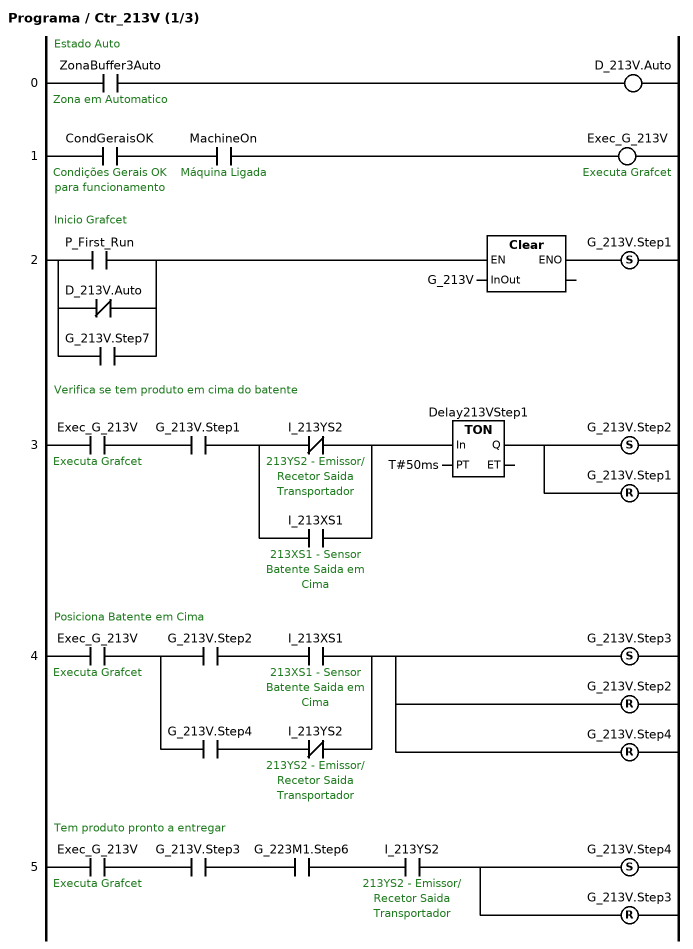
(* [picture p48: Programa / Ctr_213V, rungs 0-5] *)
(* Rung 0: Estado Auto *)
D_213V.Auto := ZonaBuffer3Auto;
(* Rung 1 *)
Exec_G_213V := CondGeraisOK AND MachineOn;
(* Rung 2: Inicio Grafcet *)
_p80 := P_First_Run OR NOT D_213V.Auto OR G_213V.Step7;
IF _p80 THEN
    Clear(InOut := G_213V);
    G_213V.Step1 := TRUE;
END_IF;
(* Rung 3: Verifica se tem produto em cima do batente *)
Delay213VStep1(In := Exec_G_213V AND G_213V.Step1 AND (NOT I_213YS2 OR I_213XS1), PT := T#50ms);
IF Delay213VStep1.Q THEN
    G_213V.Step2 := TRUE;
    G_213V.Step1 := FALSE;
END_IF;
(* Rung 4: Posiciona Batente em Cima *)
_p81 := Exec_G_213V AND ((G_213V.Step2 AND I_213XS1) OR (G_213V.Step4 AND NOT I_213YS2));
IF _p81 THEN
    G_213V.Step3 := TRUE;
    G_213V.Step2 := FALSE;
    G_213V.Step4 := FALSE;
END_IF;
(* Rung 5: Tem produto pronto a entregar *)
_p82 := Exec_G_213V AND G_213V.Step3 AND G_223M1.Step6 AND I_213YS2;
IF _p82 THEN
    G_213V.Step4 := TRUE;
    G_213V.Step3 := FALSE;
END_IF;

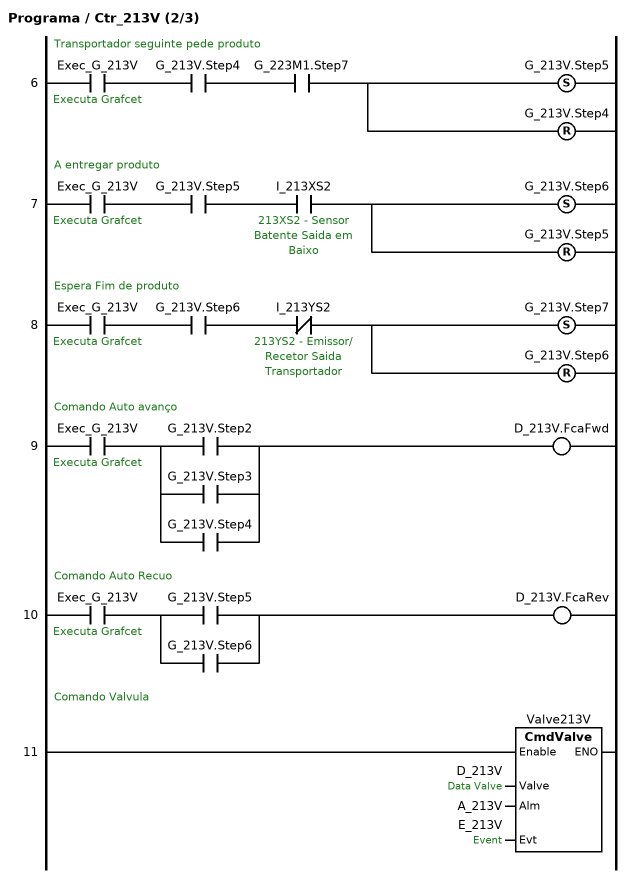
(* Rung 6: Transportador seguinte pede produto *)
_p83 := Exec_G_213V AND G_213V.Step4 AND G_223M1.Step7;
IF _p83 THEN
    G_213V.Step5 := TRUE;
    G_213V.Step4 := FALSE;
END_IF;
(* Rung 7: A entregar produto *)
_p84 := Exec_G_213V AND G_213V.Step5 AND I_213XS2;
IF _p84 THEN
    G_213V.Step6 := TRUE;
    G_213V.Step5 := FALSE;
END_IF;
(* Rung 8: Espera Fim de produto *)
_p85 := Exec_G_213V AND G_213V.Step6 AND NOT I_213YS2;
IF _p85 THEN
    G_213V.Step7 := TRUE;
    G_213V.Step6 := FALSE;
END_IF;
(* Rung 9: Comando Auto avanço *)
D_213V.FcaFwd := Exec_G_213V AND (G_213V.Step2 OR G_213V.Step3 OR G_213V.Step4);
(* Rung 10: Comando Auto Recuo *)
D_213V.FcaRev := Exec_G_213V AND (G_213V.Step5 OR G_213V.Step6);
(* Rung 11: Comando Valvula *)
Valve213V(Enable := TRUE, Valve := D_213V, Alm := A_213V, Evt := E_213V);

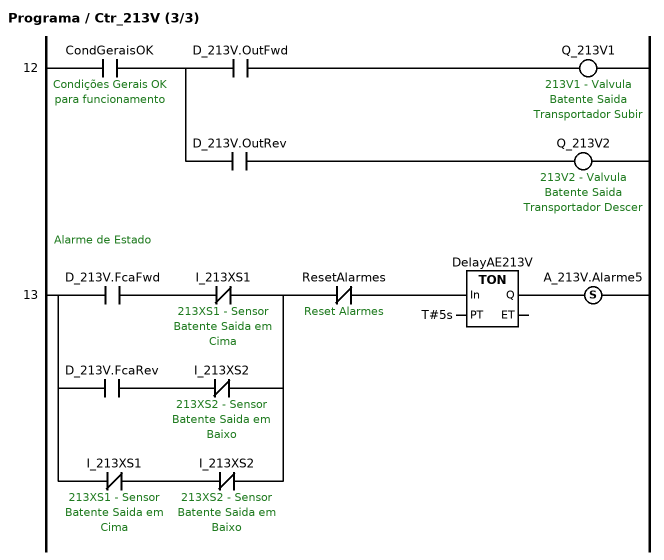
(* Rung 12 *)
Q_213V1 := CondGeraisOK AND D_213V.OutFwd;
Q_213V2 := CondGeraisOK AND D_213V.OutRev;
(* Rung 13: Alarme de Estado *)
DelayAE213V(In := ((D_213V.FcaFwd AND NOT I_213XS1) OR (D_213V.FcaRev AND NOT I_213XS2) OR (NOT I_213XS1 AND NOT I_213XS2)) AND NOT ResetAlarmes, PT := T#5s);
IF DelayAE213V.Q THEN A_213V.Alarme5 := TRUE; END_IF;

(* Section GestaoDescargaBuffers: ladder, written here as Structured Text *)

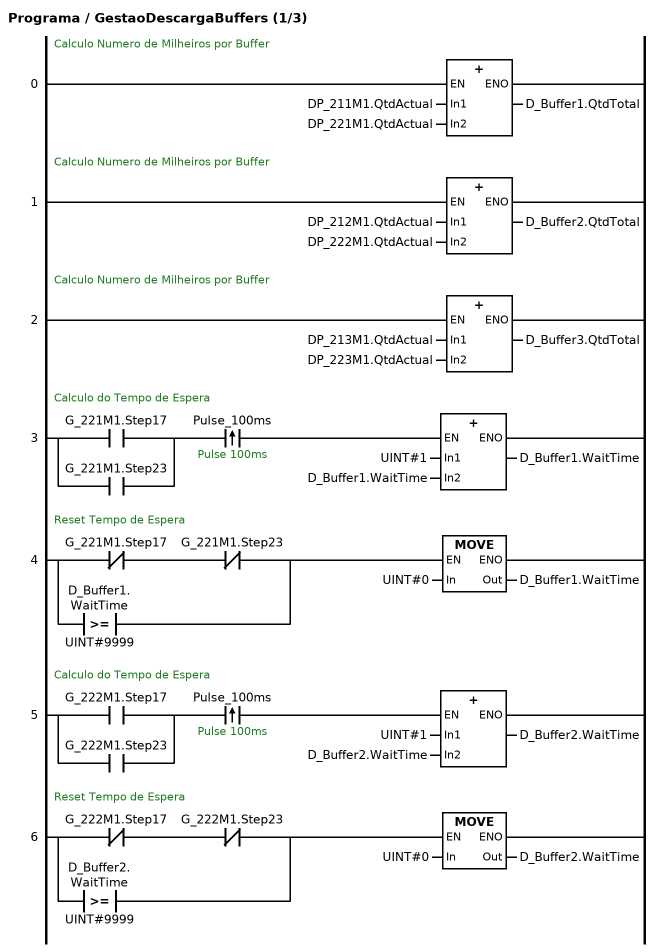
(* Rung 0: Calculo Numero de Milheiros por Buffer *)
D_Buffer1.QtdTotal := DP_211M1.QtdActual + DP_221M1.QtdActual;
(* Rung 1: Calculo Numero de Milheiros por Buffer *)
D_Buffer2.QtdTotal := DP_212M1.QtdActual + DP_222M1.QtdActual;
(* Rung 2: Calculo Numero de Milheiros por Buffer *)
D_Buffer3.QtdTotal := DP_213M1.QtdActual + DP_223M1.QtdActual;
(* Rung 3: Calculo do Tempo de Espera *)
_e86(CLK := Pulse_100ms);
IF (G_221M1.Step17 OR G_221M1.Step23) AND _e86.Q THEN
    D_Buffer1.WaitTime := UINT#1 + D_Buffer1.WaitTime;
END_IF;
(* Rung 4: Reset Tempo de Espera *)
IF (NOT G_221M1.Step17 AND NOT G_221M1.Step23) OR (D_Buffer1.WaitTime >= UINT#9999) THEN
    D_Buffer1.WaitTime := UINT#0;
END_IF;
(* Rung 5: Calculo do Tempo de Espera *)
_e87(CLK := Pulse_100ms);
IF (G_222M1.Step17 OR G_222M1.Step23) AND _e87.Q THEN
    D_Buffer2.WaitTime := UINT#1 + D_Buffer2.WaitTime;
END_IF;
(* Rung 6: Reset Tempo de Espera *)
IF (NOT G_222M1.Step17 AND NOT G_222M1.Step23) OR (D_Buffer2.WaitTime >= UINT#9999) THEN
    D_Buffer2.WaitTime := UINT#0;
END_IF;

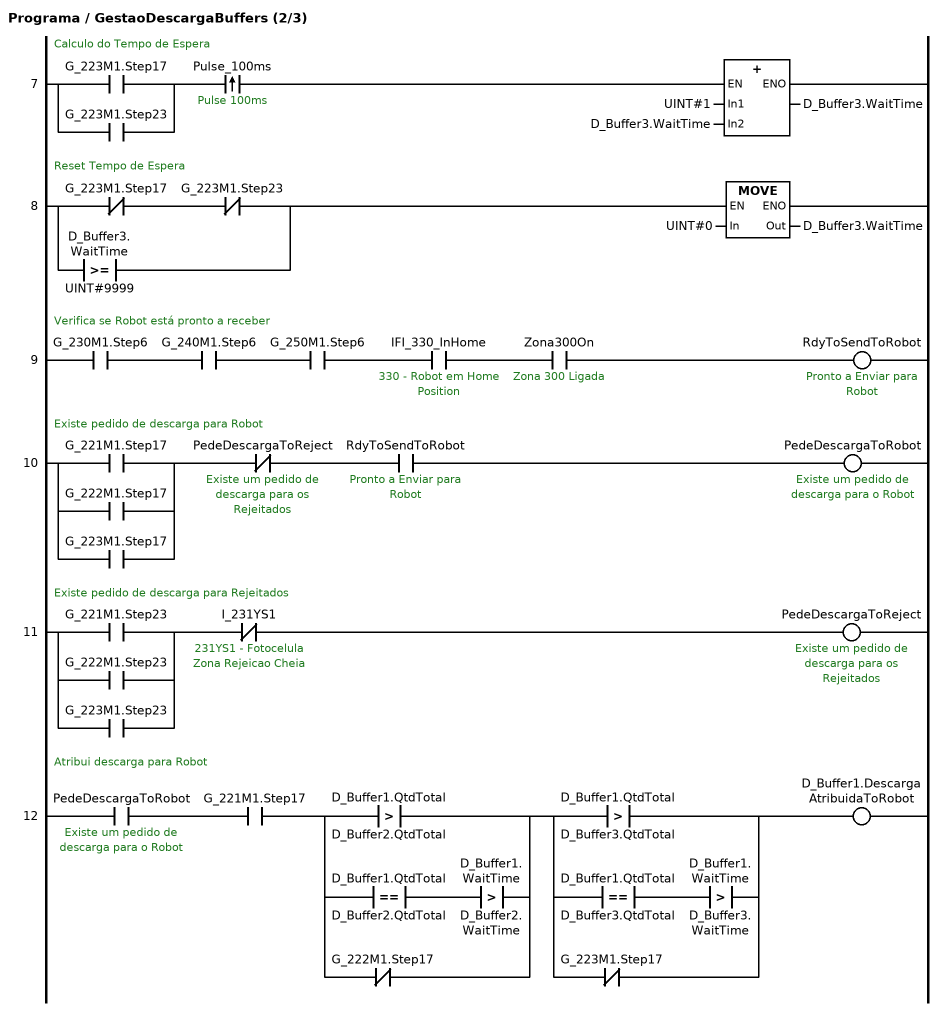
(* Rung 7: Calculo do Tempo de Espera *)
_e88(CLK := Pulse_100ms);
IF (G_223M1.Step17 OR G_223M1.Step23) AND _e88.Q THEN
    D_Buffer3.WaitTime := UINT#1 + D_Buffer3.WaitTime;
END_IF;
(* Rung 8: Reset Tempo de Espera *)
IF (NOT G_223M1.Step17 AND NOT G_223M1.Step23) OR (D_Buffer3.WaitTime >= UINT#9999) THEN
    D_Buffer3.WaitTime := UINT#0;
END_IF;
(* Rung 9: Verifica se Robot está pronto a receber *)
RdyToSendToRobot := G_230M1.Step6 AND G_240M1.Step6 AND G_250M1.Step6 AND IFI_330_InHome AND Zona300On;
(* Rung 10: Existe pedido de descarga para Robot *)
PedeDescargaToRobot := (G_221M1.Step17 OR G_222M1.Step17 OR G_223M1.Step17) AND NOT PedeDescargaToReject AND RdyToSendToRobot;
(* Rung 11: Existe pedido de descarga para Rejeitados *)
PedeDescargaToReject := (G_221M1.Step23 OR G_222M1.Step23 OR G_223M1.Step23) AND NOT I_231YS1;
(* Rung 12: Atribui descarga para Robot *)
D_Buffer1.DescargaAtribuidaToRobot := PedeDescargaToRobot AND G_221M1.Step17 AND ((D_Buffer1.QtdTotal > D_Buffer2.QtdTotal) OR ((D_Buffer1.QtdTotal = D_Buffer2.QtdTotal) AND (D_Buffer1.WaitTime > D_Buffer2.WaitTime)) OR NOT G_222M1.Step17) AND ((D_Buffer1.QtdTotal > D_Buffer3.QtdTotal) OR ((D_Buffer1.QtdTotal = D_Buffer3.QtdTotal) AND (D_Buffer1.WaitTime > D_Buffer3.WaitTime)) OR NOT G_223M1.Step17);

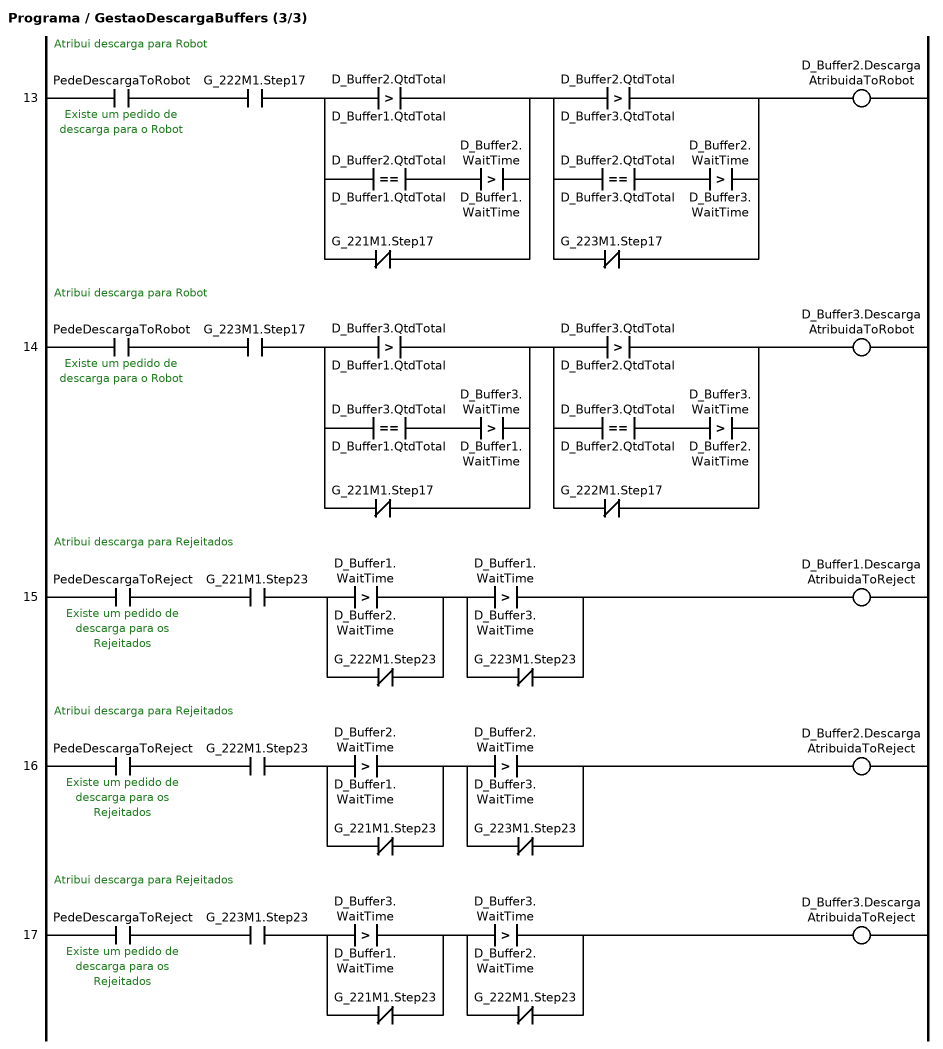
(* Rung 13: Atribui descarga para Robot *)
D_Buffer2.DescargaAtribuidaToRobot := PedeDescargaToRobot AND G_222M1.Step17 AND ((D_Buffer2.QtdTotal > D_Buffer1.QtdTotal) OR ((D_Buffer2.QtdTotal = D_Buffer1.QtdTotal) AND (D_Buffer2.WaitTime > D_Buffer1.WaitTime)) OR NOT G_221M1.Step17) AND ((D_Buffer2.QtdTotal > D_Buffer3.QtdTotal) OR ((D_Buffer2.QtdTotal = D_Buffer3.QtdTotal) AND (D_Buffer2.WaitTime > D_Buffer3.WaitTime)) OR NOT G_223M1.Step17);
(* Rung 14: Atribui descarga para Robot *)
D_Buffer3.DescargaAtribuidaToRobot := PedeDescargaToRobot AND G_223M1.Step17 AND ((D_Buffer3.QtdTotal > D_Buffer1.QtdTotal) OR ((D_Buffer3.QtdTotal = D_Buffer1.QtdTotal) AND (D_Buffer3.WaitTime > D_Buffer1.WaitTime)) OR NOT G_221M1.Step17) AND ((D_Buffer3.QtdTotal > D_Buffer2.QtdTotal) OR ((D_Buffer3.QtdTotal = D_Buffer2.QtdTotal) AND (D_Buffer3.WaitTime > D_Buffer2.WaitTime)) OR NOT G_222M1.Step17);
(* Rung 15: Atribui descarga para Rejeitados *)
D_Buffer1.DescargaAtribuidaToReject := PedeDescargaToReject AND G_221M1.Step23 AND ((D_Buffer1.WaitTime > D_Buffer2.WaitTime) OR NOT G_222M1.Step23) AND ((D_Buffer1.WaitTime > D_Buffer3.WaitTime) OR NOT G_223M1.Step23);
(* Rung 16: Atribui descarga para Rejeitados *)
D_Buffer2.DescargaAtribuidaToReject := PedeDescargaToReject AND G_222M1.Step23 AND ((D_Buffer2.WaitTime > D_Buffer1.WaitTime) OR NOT G_221M1.Step23) AND ((D_Buffer2.WaitTime > D_Buffer3.WaitTime) OR NOT G_223M1.Step23);
(* Rung 17: Atribui descarga para Rejeitados *)
D_Buffer3.DescargaAtribuidaToReject := PedeDescargaToReject AND G_223M1.Step23 AND ((D_Buffer3.WaitTime > D_Buffer1.WaitTime) OR NOT G_221M1.Step23) AND ((D_Buffer3.WaitTime > D_Buffer2.WaitTime) OR NOT G_222M1.Step23);

(* Section Ctr_221M1: ladder, written here as Structured Text *)

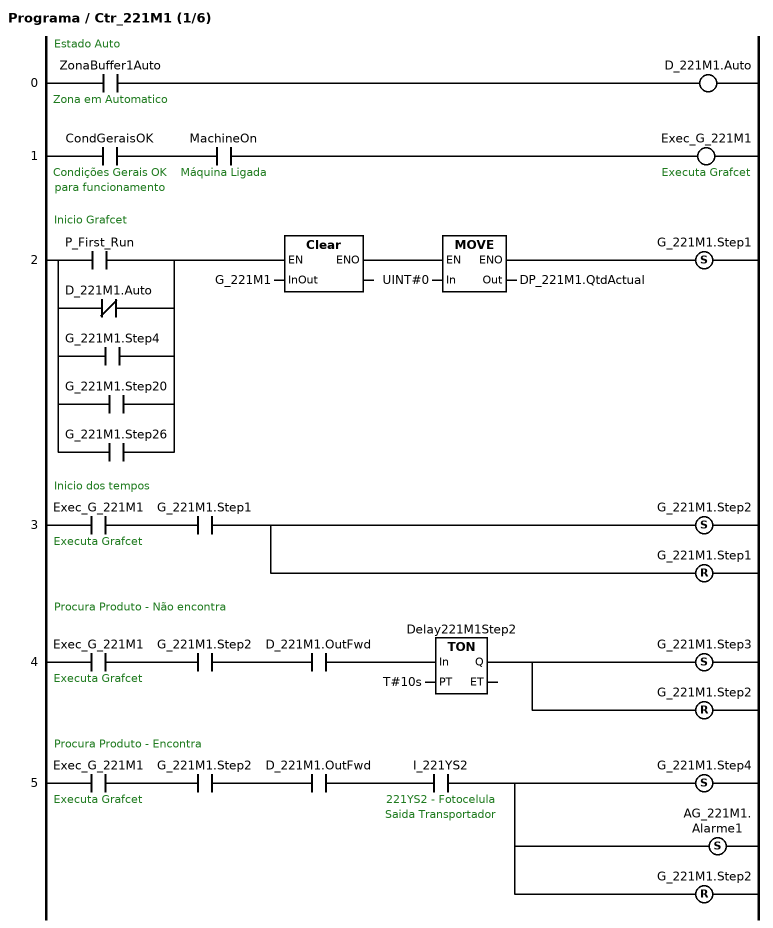
(* Rung 0: Estado Auto *)
D_221M1.Auto := ZonaBuffer1Auto;
(* Rung 1 *)
Exec_G_221M1 := CondGeraisOK AND MachineOn;
(* Rung 2: Inicio Grafcet *)
_p89 := P_First_Run OR NOT D_221M1.Auto OR G_221M1.Step4 OR G_221M1.Step20 OR G_221M1.Step26;
IF _p89 THEN
    Clear(InOut := G_221M1);
    DP_221M1.QtdActual := UINT#0;
    G_221M1.Step1 := TRUE;
END_IF;
(* Rung 3: Inicio dos tempos *)
_p90 := Exec_G_221M1 AND G_221M1.Step1;
IF _p90 THEN
    G_221M1.Step2 := TRUE;
    G_221M1.Step1 := FALSE;
END_IF;
(* Rung 4: Procura Produto - Não encontra *)
Delay221M1Step2(In := Exec_G_221M1 AND G_221M1.Step2 AND D_221M1.OutFwd, PT := T#10s);
IF Delay221M1Step2.Q THEN
    G_221M1.Step3 := TRUE;
    G_221M1.Step2 := FALSE;
END_IF;
(* Rung 5: Procura Produto - Encontra *)
_p91 := Exec_G_221M1 AND G_221M1.Step2 AND D_221M1.OutFwd AND I_221YS2;
IF _p91 THEN
    G_221M1.Step4 := TRUE;
    AG_221M1.Alarme1 := TRUE;
    G_221M1.Step2 := FALSE;
END_IF;

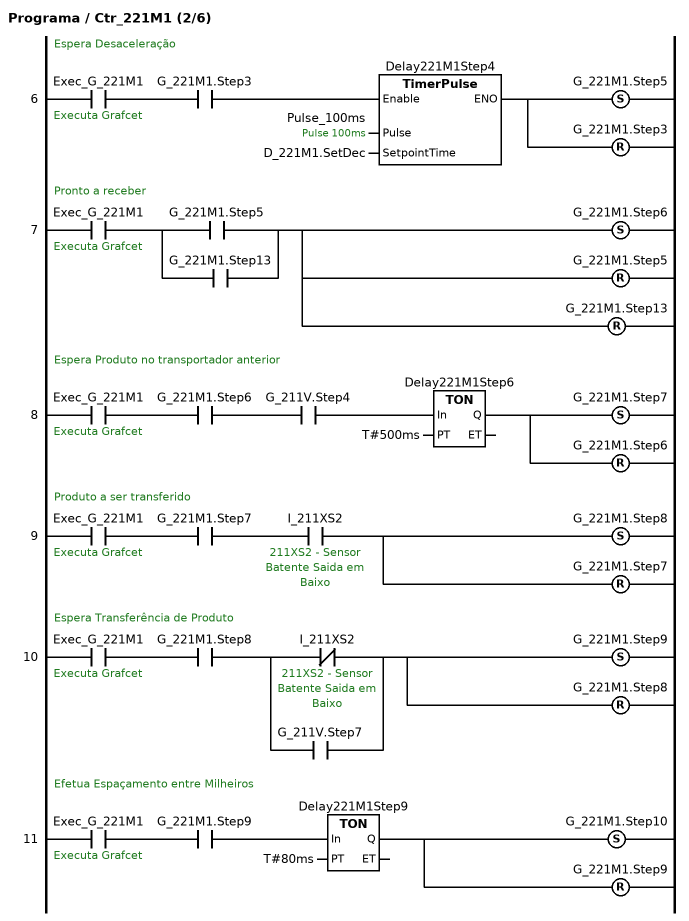
(* Rung 6: Espera Desaceleração *)
Delay221M1Step4(Enable := Exec_G_221M1 AND G_221M1.Step3, Pulse := Pulse_100ms, SetpointTime := D_221M1.SetDec);
IF Delay221M1Step4.ENO THEN
    G_221M1.Step5 := TRUE;
    G_221M1.Step3 := FALSE;
END_IF;
(* Rung 7: Pronto a receber *)
_p92 := Exec_G_221M1 AND (G_221M1.Step5 OR G_221M1.Step13);
IF _p92 THEN
    G_221M1.Step6 := TRUE;
    G_221M1.Step5 := FALSE;
    G_221M1.Step13 := FALSE;
END_IF;
(* Rung 8: Espera Produto no transportador anterior *)
Delay221M1Step6(In := Exec_G_221M1 AND G_221M1.Step6 AND G_211V.Step4, PT := T#500ms);
IF Delay221M1Step6.Q THEN
    G_221M1.Step7 := TRUE;
    G_221M1.Step6 := FALSE;
END_IF;
(* Rung 9: Produto a ser transferido *)
_p93 := Exec_G_221M1 AND G_221M1.Step7 AND I_211XS2;
IF _p93 THEN
    G_221M1.Step8 := TRUE;
    G_221M1.Step7 := FALSE;
END_IF;
(* Rung 10: Espera Transferência de Produto *)
_p94 := Exec_G_221M1 AND G_221M1.Step8 AND (NOT I_211XS2 OR G_211V.Step7);
IF _p94 THEN
    G_221M1.Step9 := TRUE;
    G_221M1.Step8 := FALSE;
END_IF;
(* Rung 11: Efetua Espaçamento entre Milheiros *)
Delay221M1Step9(In := Exec_G_221M1 AND G_221M1.Step9, PT := T#80ms);
IF Delay221M1Step9.Q THEN
    G_221M1.Step10 := TRUE;
    G_221M1.Step9 := FALSE;
END_IF;

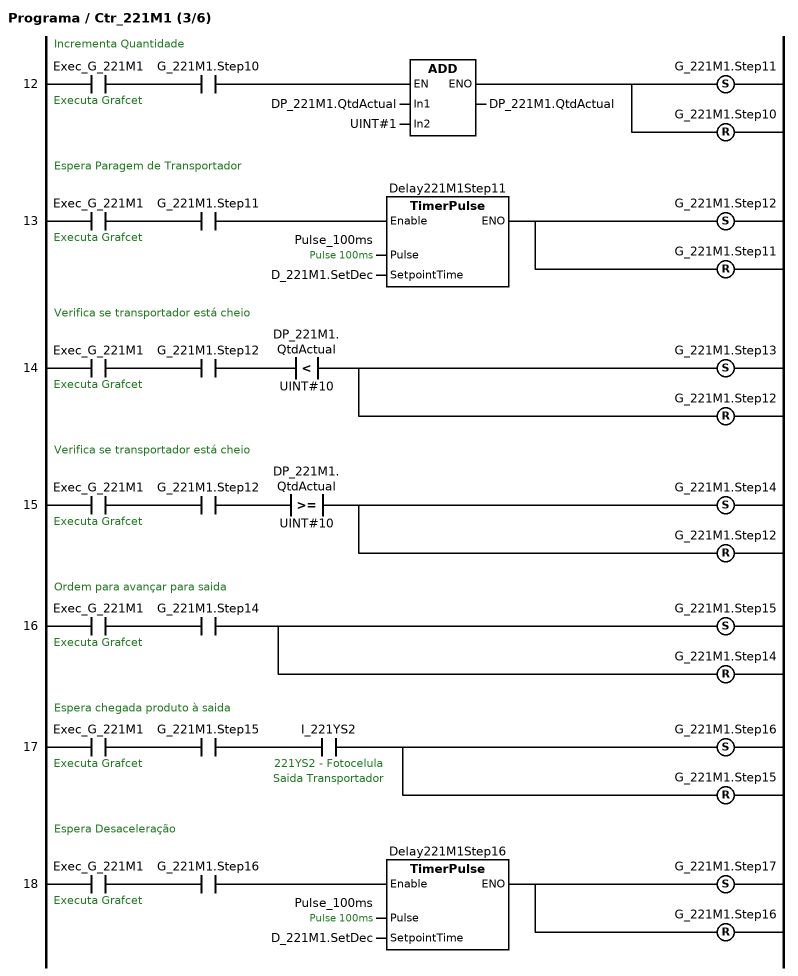
(* Rung 12: Incrementa Quantidade *)
IF Exec_G_221M1 AND G_221M1.Step10 THEN DP_221M1.QtdActual := DP_221M1.QtdActual + UINT#1; END_IF;
_p95 := Exec_G_221M1 AND G_221M1.Step10;
IF _p95 THEN
    G_221M1.Step11 := TRUE;
    G_221M1.Step10 := FALSE;
END_IF;
(* Rung 13: Espera Paragem de Transportador *)
Delay221M1Step11(Enable := Exec_G_221M1 AND G_221M1.Step11, Pulse := Pulse_100ms, SetpointTime := D_221M1.SetDec);
IF Delay221M1Step11.ENO THEN
    G_221M1.Step12 := TRUE;
    G_221M1.Step11 := FALSE;
END_IF;
(* Rung 14: Verifica se transportador está cheio *)
_p96 := Exec_G_221M1 AND G_221M1.Step12 AND (DP_221M1.QtdActual < UINT#10);
IF _p96 THEN
    G_221M1.Step13 := TRUE;
    G_221M1.Step12 := FALSE;
END_IF;
(* Rung 15: Verifica se transportador está cheio *)
_p97 := Exec_G_221M1 AND G_221M1.Step12 AND (DP_221M1.QtdActual >= UINT#10);
IF _p97 THEN
    G_221M1.Step14 := TRUE;
    G_221M1.Step12 := FALSE;
END_IF;
(* Rung 16: Ordem para avançar para saida *)
_p98 := Exec_G_221M1 AND G_221M1.Step14;
IF _p98 THEN
    G_221M1.Step15 := TRUE;
    G_221M1.Step14 := FALSE;
END_IF;
(* Rung 17: Espera chegada produto à saida *)
_p99 := Exec_G_221M1 AND G_221M1.Step15 AND I_221YS2;
IF _p99 THEN
    G_221M1.Step16 := TRUE;
    G_221M1.Step15 := FALSE;
END_IF;
(* Rung 18: Espera Desaceleração *)
Delay221M1Step16(Enable := Exec_G_221M1 AND G_221M1.Step16, Pulse := Pulse_100ms, SetpointTime := D_221M1.SetDec);
IF Delay221M1Step16.ENO THEN
    G_221M1.Step17 := TRUE;
    G_221M1.Step16 := FALSE;
END_IF;

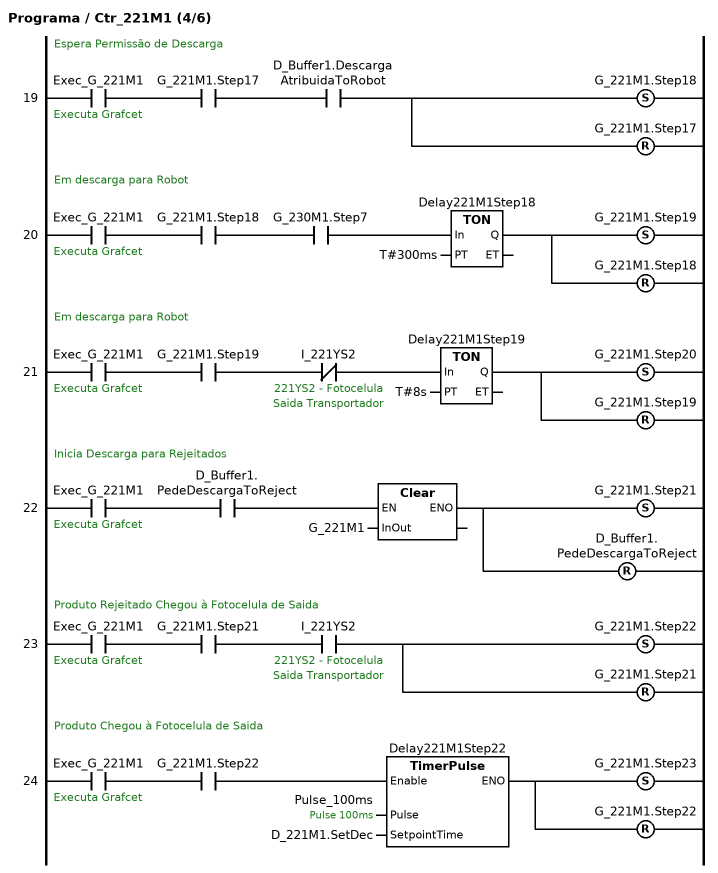
(* Rung 19: Espera Permissão de Descarga *)
_p100 := Exec_G_221M1 AND G_221M1.Step17 AND D_Buffer1.DescargaAtribuidaToRobot;
IF _p100 THEN
    G_221M1.Step18 := TRUE;
    G_221M1.Step17 := FALSE;
END_IF;
(* Rung 20: Em descarga para Robot *)
Delay221M1Step18(In := Exec_G_221M1 AND G_221M1.Step18 AND G_230M1.Step7, PT := T#300ms);
IF Delay221M1Step18.Q THEN
    G_221M1.Step19 := TRUE;
    G_221M1.Step18 := FALSE;
END_IF;
(* Rung 21: Em descarga para Robot *)
Delay221M1Step19(In := Exec_G_221M1 AND G_221M1.Step19 AND NOT I_221YS2, PT := T#8s);
IF Delay221M1Step19.Q THEN
    G_221M1.Step20 := TRUE;
    G_221M1.Step19 := FALSE;
END_IF;
(* Rung 22: Inicia Descarga para Rejeitados *)
IF Exec_G_221M1 AND D_Buffer1.PedeDescargaToReject THEN
    Clear(InOut := G_221M1);
    G_221M1.Step21 := TRUE;
    D_Buffer1.PedeDescargaToReject := FALSE;
END_IF;
(* Rung 23: Produto Rejeitado Chegou à Fotocelula de Saida *)
_p101 := Exec_G_221M1 AND G_221M1.Step21 AND I_221YS2;
IF _p101 THEN
    G_221M1.Step22 := TRUE;
    G_221M1.Step21 := FALSE;
END_IF;
(* Rung 24: Produto Chegou à Fotocelula de Saida *)
Delay221M1Step22(Enable := Exec_G_221M1 AND G_221M1.Step22, Pulse := Pulse_100ms, SetpointTime := D_221M1.SetDec);
IF Delay221M1Step22.ENO THEN
    G_221M1.Step23 := TRUE;
    G_221M1.Step22 := FALSE;
END_IF;

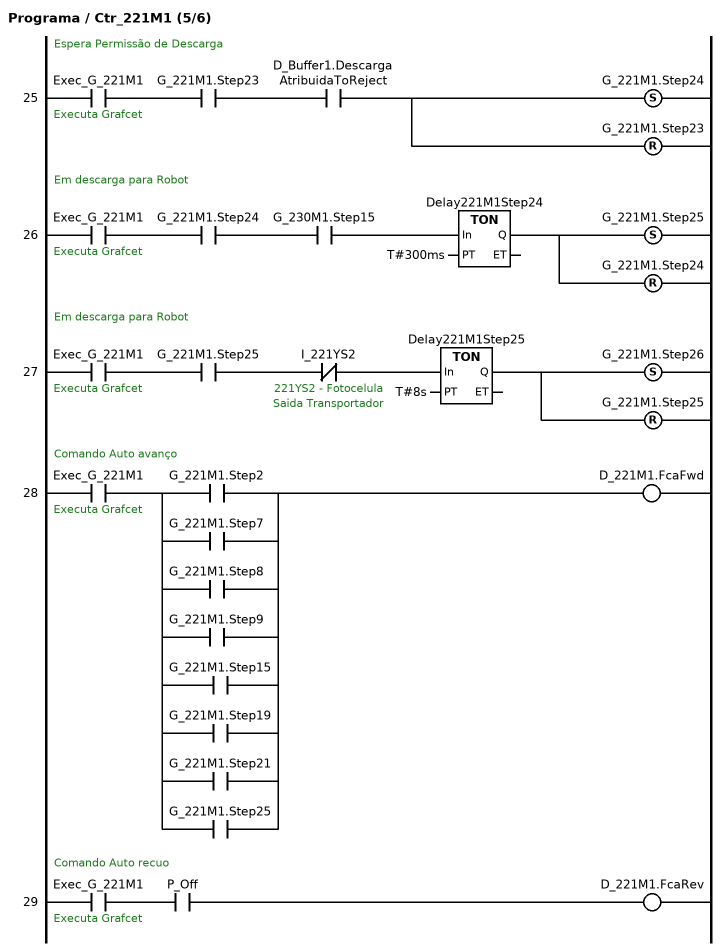
(* Rung 25: Espera Permissão de Descarga *)
_p102 := Exec_G_221M1 AND G_221M1.Step23 AND D_Buffer1.DescargaAtribuidaToReject;
IF _p102 THEN
    G_221M1.Step24 := TRUE;
    G_221M1.Step23 := FALSE;
END_IF;
(* Rung 26: Em descarga para Robot *)
Delay221M1Step24(In := Exec_G_221M1 AND G_221M1.Step24 AND G_230M1.Step15, PT := T#300ms);
IF Delay221M1Step24.Q THEN
    G_221M1.Step25 := TRUE;
    G_221M1.Step24 := FALSE;
END_IF;
(* Rung 27: Em descarga para Robot *)
Delay221M1Step25(In := Exec_G_221M1 AND G_221M1.Step25 AND NOT I_221YS2, PT := T#8s);
IF Delay221M1Step25.Q THEN
    G_221M1.Step26 := TRUE;
    G_221M1.Step25 := FALSE;
END_IF;
(* Rung 28: Comando Auto avanço *)
D_221M1.FcaFwd := Exec_G_221M1 AND (G_221M1.Step2 OR G_221M1.Step7 OR G_221M1.Step8 OR G_221M1.Step9 OR G_221M1.Step15 OR G_221M1.Step19 OR G_221M1.Step21 OR G_221M1.Step25);
(* Rung 29: Comando Auto recuo *)
D_221M1.FcaRev := Exec_G_221M1 AND P_Off;

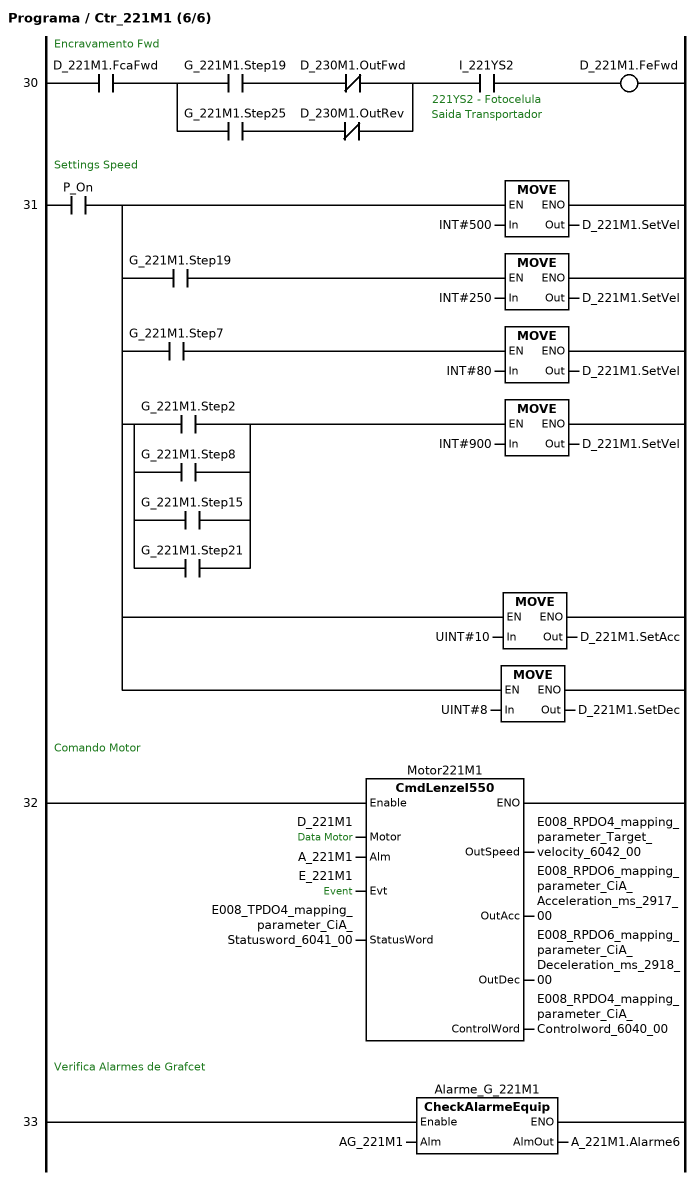
(* Rung 30: Encravamento Fwd *)
D_221M1.FeFwd := D_221M1.FcaFwd AND ((G_221M1.Step19 AND NOT D_230M1.OutFwd) OR (G_221M1.Step25 AND NOT D_230M1.OutRev)) AND I_221YS2;
(* Rung 31: Settings Speed *)
IF P_On THEN D_221M1.SetVel := INT#500; END_IF;
IF P_On AND G_221M1.Step19 THEN D_221M1.SetVel := INT#250; END_IF;
IF P_On AND G_221M1.Step7 THEN D_221M1.SetVel := INT#80; END_IF;
IF P_On AND (G_221M1.Step2 OR G_221M1.Step8 OR G_221M1.Step15 OR G_221M1.Step21) THEN
    D_221M1.SetVel := INT#900;
END_IF;
IF P_On THEN
    D_221M1.SetAcc := UINT#10;
    D_221M1.SetDec := UINT#8;
END_IF;
(* Rung 32: Comando Motor *)
Motor221M1(Enable := TRUE, Motor := D_221M1, Alm := A_221M1, Evt := E_221M1, StatusWord := E008_TPDO4_mapping_parameter_CiA_Statusword_6041_00, OutSpeed => E008_RPDO4_mapping_parameter_Target_velocity_6042_00, OutAcc => E008_RPDO6_mapping_parameter_CiA_Acceleration_ms_2917_00, OutDec => E008_RPDO6_mapping_parameter_CiA_Deceleration_ms_2918_00, ControlWord => E008_RPDO4_mapping_parameter_CiA_Controlword_6040_00);
(* Rung 33: Verifica Alarmes de Grafcet *)
Alarme_G_221M1(Enable := TRUE, Alm := AG_221M1, AlmOut => A_221M1.Alarme6);

(* Section Ctr_222M1: ladder, written here as Structured Text *)

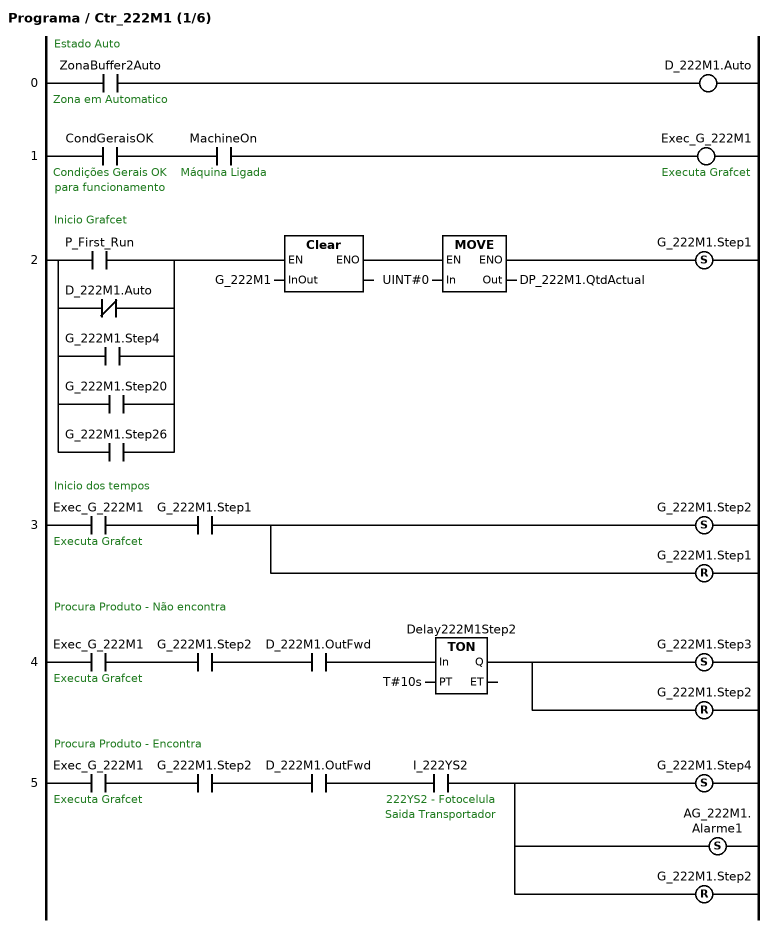
(* Rung 0: Estado Auto *)
D_222M1.Auto := ZonaBuffer2Auto;
(* Rung 1 *)
Exec_G_222M1 := CondGeraisOK AND MachineOn;
(* Rung 2: Inicio Grafcet *)
_p103 := P_First_Run OR NOT D_222M1.Auto OR G_222M1.Step4 OR G_222M1.Step20 OR G_222M1.Step26;
IF _p103 THEN
    Clear(InOut := G_222M1);
    DP_222M1.QtdActual := UINT#0;
    G_222M1.Step1 := TRUE;
END_IF;
(* Rung 3: Inicio dos tempos *)
_p104 := Exec_G_222M1 AND G_222M1.Step1;
IF _p104 THEN
    G_222M1.Step2 := TRUE;
    G_222M1.Step1 := FALSE;
END_IF;
(* Rung 4: Procura Produto - Não encontra *)
Delay222M1Step2(In := Exec_G_222M1 AND G_222M1.Step2 AND D_222M1.OutFwd, PT := T#10s);
IF Delay222M1Step2.Q THEN
    G_222M1.Step3 := TRUE;
    G_222M1.Step2 := FALSE;
END_IF;
(* Rung 5: Procura Produto - Encontra *)
_p105 := Exec_G_222M1 AND G_222M1.Step2 AND D_222M1.OutFwd AND I_222YS2;
IF _p105 THEN
    G_222M1.Step4 := TRUE;
    AG_222M1.Alarme1 := TRUE;
    G_222M1.Step2 := FALSE;
END_IF;

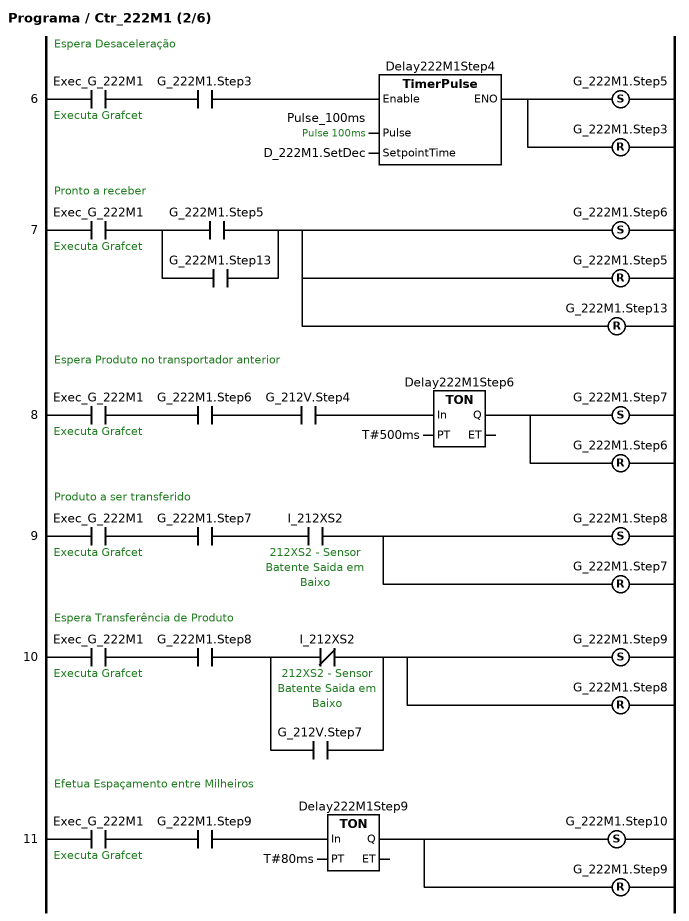
(* Rung 6: Espera Desaceleração *)
Delay222M1Step4(Enable := Exec_G_222M1 AND G_222M1.Step3, Pulse := Pulse_100ms, SetpointTime := D_222M1.SetDec);
IF Delay222M1Step4.ENO THEN
    G_222M1.Step5 := TRUE;
    G_222M1.Step3 := FALSE;
END_IF;
(* Rung 7: Pronto a receber *)
_p106 := Exec_G_222M1 AND (G_222M1.Step5 OR G_222M1.Step13);
IF _p106 THEN
    G_222M1.Step6 := TRUE;
    G_222M1.Step5 := FALSE;
    G_222M1.Step13 := FALSE;
END_IF;
(* Rung 8: Espera Produto no transportador anterior *)
Delay222M1Step6(In := Exec_G_222M1 AND G_222M1.Step6 AND G_212V.Step4, PT := T#500ms);
IF Delay222M1Step6.Q THEN
    G_222M1.Step7 := TRUE;
    G_222M1.Step6 := FALSE;
END_IF;
(* Rung 9: Produto a ser transferido *)
_p107 := Exec_G_222M1 AND G_222M1.Step7 AND I_212XS2;
IF _p107 THEN
    G_222M1.Step8 := TRUE;
    G_222M1.Step7 := FALSE;
END_IF;
(* Rung 10: Espera Transferência de Produto *)
_p108 := Exec_G_222M1 AND G_222M1.Step8 AND (NOT I_212XS2 OR G_212V.Step7);
IF _p108 THEN
    G_222M1.Step9 := TRUE;
    G_222M1.Step8 := FALSE;
END_IF;
(* Rung 11: Efetua Espaçamento entre Milheiros *)
Delay222M1Step9(In := Exec_G_222M1 AND G_222M1.Step9, PT := T#80ms);
IF Delay222M1Step9.Q THEN
    G_222M1.Step10 := TRUE;
    G_222M1.Step9 := FALSE;
END_IF;

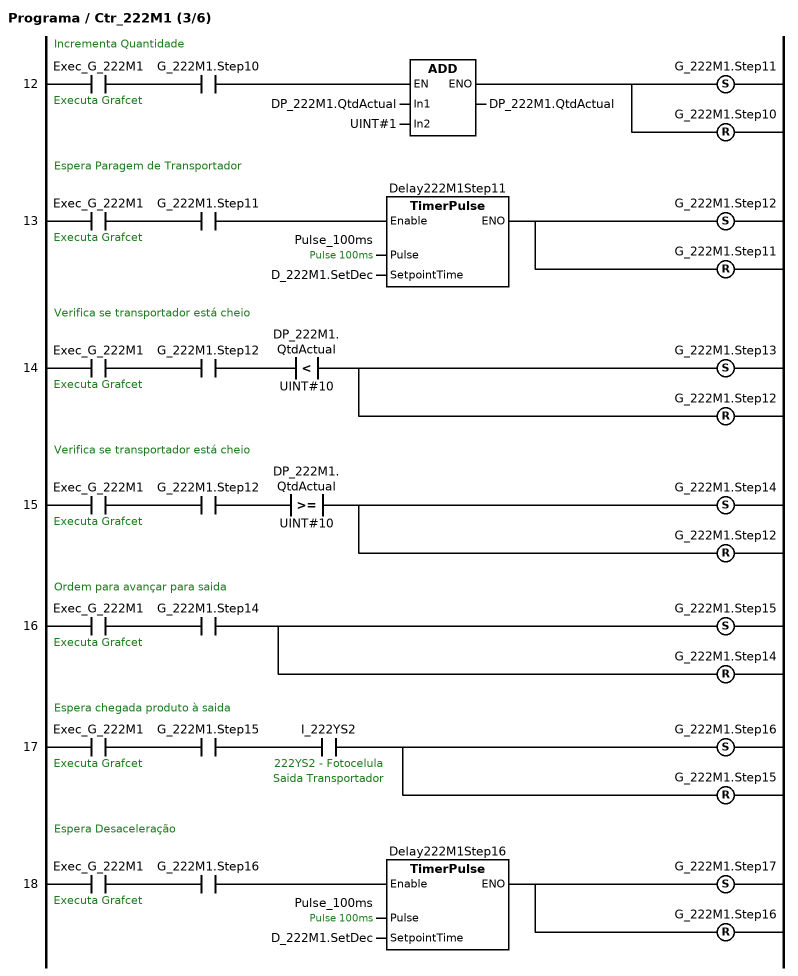
(* Rung 12: Incrementa Quantidade *)
IF Exec_G_222M1 AND G_222M1.Step10 THEN DP_222M1.QtdActual := DP_222M1.QtdActual + UINT#1; END_IF;
_p109 := Exec_G_222M1 AND G_222M1.Step10;
IF _p109 THEN
    G_222M1.Step11 := TRUE;
    G_222M1.Step10 := FALSE;
END_IF;
(* Rung 13: Espera Paragem de Transportador *)
Delay222M1Step11(Enable := Exec_G_222M1 AND G_222M1.Step11, Pulse := Pulse_100ms, SetpointTime := D_222M1.SetDec);
IF Delay222M1Step11.ENO THEN
    G_222M1.Step12 := TRUE;
    G_222M1.Step11 := FALSE;
END_IF;
(* Rung 14: Verifica se transportador está cheio *)
_p110 := Exec_G_222M1 AND G_222M1.Step12 AND (DP_222M1.QtdActual < UINT#10);
IF _p110 THEN
    G_222M1.Step13 := TRUE;
    G_222M1.Step12 := FALSE;
END_IF;
(* Rung 15: Verifica se transportador está cheio *)
_p111 := Exec_G_222M1 AND G_222M1.Step12 AND (DP_222M1.QtdActual >= UINT#10);
IF _p111 THEN
    G_222M1.Step14 := TRUE;
    G_222M1.Step12 := FALSE;
END_IF;
(* Rung 16: Ordem para avançar para saida *)
_p112 := Exec_G_222M1 AND G_222M1.Step14;
IF _p112 THEN
    G_222M1.Step15 := TRUE;
    G_222M1.Step14 := FALSE;
END_IF;
(* Rung 17: Espera chegada produto à saida *)
_p113 := Exec_G_222M1 AND G_222M1.Step15 AND I_222YS2;
IF _p113 THEN
    G_222M1.Step16 := TRUE;
    G_222M1.Step15 := FALSE;
END_IF;
(* Rung 18: Espera Desaceleração *)
Delay222M1Step16(Enable := Exec_G_222M1 AND G_222M1.Step16, Pulse := Pulse_100ms, SetpointTime := D_222M1.SetDec);
IF Delay222M1Step16.ENO THEN
    G_222M1.Step17 := TRUE;
    G_222M1.Step16 := FALSE;
END_IF;

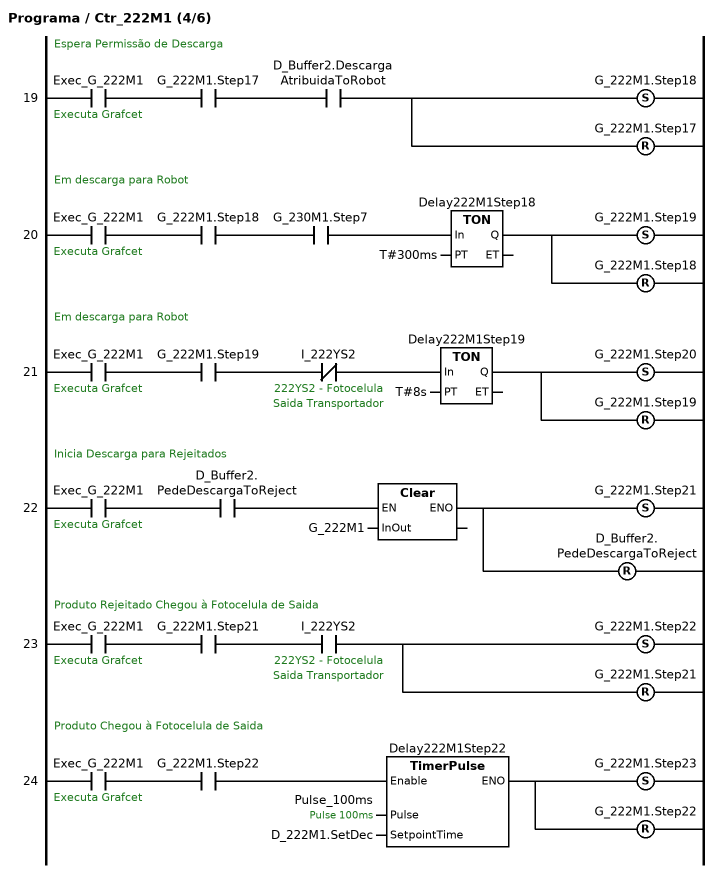
(* Rung 19: Espera Permissão de Descarga *)
_p114 := Exec_G_222M1 AND G_222M1.Step17 AND D_Buffer2.DescargaAtribuidaToRobot;
IF _p114 THEN
    G_222M1.Step18 := TRUE;
    G_222M1.Step17 := FALSE;
END_IF;
(* Rung 20: Em descarga para Robot *)
Delay222M1Step18(In := Exec_G_222M1 AND G_222M1.Step18 AND G_230M1.Step7, PT := T#300ms);
IF Delay222M1Step18.Q THEN
    G_222M1.Step19 := TRUE;
    G_222M1.Step18 := FALSE;
END_IF;
(* Rung 21: Em descarga para Robot *)
Delay222M1Step19(In := Exec_G_222M1 AND G_222M1.Step19 AND NOT I_222YS2, PT := T#8s);
IF Delay222M1Step19.Q THEN
    G_222M1.Step20 := TRUE;
    G_222M1.Step19 := FALSE;
END_IF;
(* Rung 22: Inicia Descarga para Rejeitados *)
IF Exec_G_222M1 AND D_Buffer2.PedeDescargaToReject THEN
    Clear(InOut := G_222M1);
    G_222M1.Step21 := TRUE;
    D_Buffer2.PedeDescargaToReject := FALSE;
END_IF;
(* Rung 23: Produto Rejeitado Chegou à Fotocelula de Saida *)
_p115 := Exec_G_222M1 AND G_222M1.Step21 AND I_222YS2;
IF _p115 THEN
    G_222M1.Step22 := TRUE;
    G_222M1.Step21 := FALSE;
END_IF;
(* Rung 24: Produto Chegou à Fotocelula de Saida *)
Delay222M1Step22(Enable := Exec_G_222M1 AND G_222M1.Step22, Pulse := Pulse_100ms, SetpointTime := D_222M1.SetDec);
IF Delay222M1Step22.ENO THEN
    G_222M1.Step23 := TRUE;
    G_222M1.Step22 := FALSE;
END_IF;

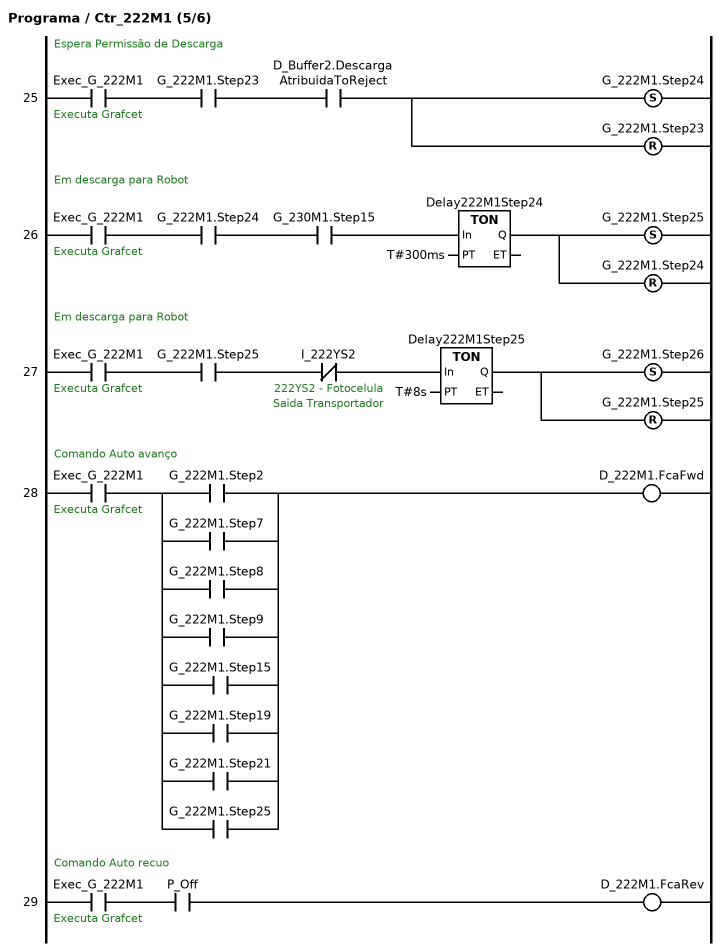
(* Rung 25: Espera Permissão de Descarga *)
_p116 := Exec_G_222M1 AND G_222M1.Step23 AND D_Buffer2.DescargaAtribuidaToReject;
IF _p116 THEN
    G_222M1.Step24 := TRUE;
    G_222M1.Step23 := FALSE;
END_IF;
(* Rung 26: Em descarga para Robot *)
Delay222M1Step24(In := Exec_G_222M1 AND G_222M1.Step24 AND G_230M1.Step15, PT := T#300ms);
IF Delay222M1Step24.Q THEN
    G_222M1.Step25 := TRUE;
    G_222M1.Step24 := FALSE;
END_IF;
(* Rung 27: Em descarga para Robot *)
Delay222M1Step25(In := Exec_G_222M1 AND G_222M1.Step25 AND NOT I_222YS2, PT := T#8s);
IF Delay222M1Step25.Q THEN
    G_222M1.Step26 := TRUE;
    G_222M1.Step25 := FALSE;
END_IF;
(* Rung 28: Comando Auto avanço *)
D_222M1.FcaFwd := Exec_G_222M1 AND (G_222M1.Step2 OR G_222M1.Step7 OR G_222M1.Step8 OR G_222M1.Step9 OR G_222M1.Step15 OR G_222M1.Step19 OR G_222M1.Step21 OR G_222M1.Step25);
(* Rung 29: Comando Auto recuo *)
D_222M1.FcaRev := Exec_G_222M1 AND P_Off;

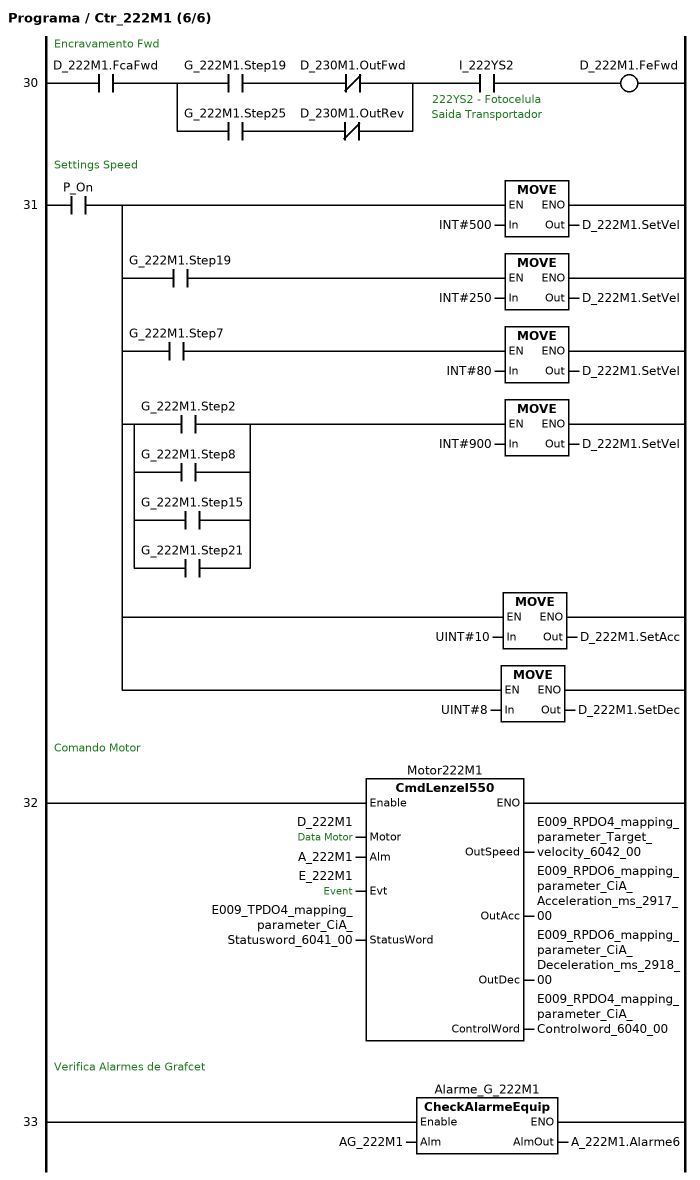
(* Rung 30: Encravamento Fwd *)
D_222M1.FeFwd := D_222M1.FcaFwd AND ((G_222M1.Step19 AND NOT D_230M1.OutFwd) OR (G_222M1.Step25 AND NOT D_230M1.OutRev)) AND I_222YS2;
(* Rung 31: Settings Speed *)
IF P_On THEN D_222M1.SetVel := INT#500; END_IF;
IF P_On AND G_222M1.Step19 THEN D_222M1.SetVel := INT#250; END_IF;
IF P_On AND G_222M1.Step7 THEN D_222M1.SetVel := INT#80; END_IF;
IF P_On AND (G_222M1.Step2 OR G_222M1.Step8 OR G_222M1.Step15 OR G_222M1.Step21) THEN
    D_222M1.SetVel := INT#900;
END_IF;
IF P_On THEN
    D_222M1.SetAcc := UINT#10;
    D_222M1.SetDec := UINT#8;
END_IF;
(* Rung 32: Comando Motor *)
Motor222M1(Enable := TRUE, Motor := D_222M1, Alm := A_222M1, Evt := E_222M1, StatusWord := E009_TPDO4_mapping_parameter_CiA_Statusword_6041_00, OutSpeed => E009_RPDO4_mapping_parameter_Target_velocity_6042_00, OutAcc => E009_RPDO6_mapping_parameter_CiA_Acceleration_ms_2917_00, OutDec => E009_RPDO6_mapping_parameter_CiA_Deceleration_ms_2918_00, ControlWord => E009_RPDO4_mapping_parameter_CiA_Controlword_6040_00);
(* Rung 33: Verifica Alarmes de Grafcet *)
Alarme_G_222M1(Enable := TRUE, Alm := AG_222M1, AlmOut => A_222M1.Alarme6);

(* Section Ctr_223M1: ladder, written here as Structured Text *)

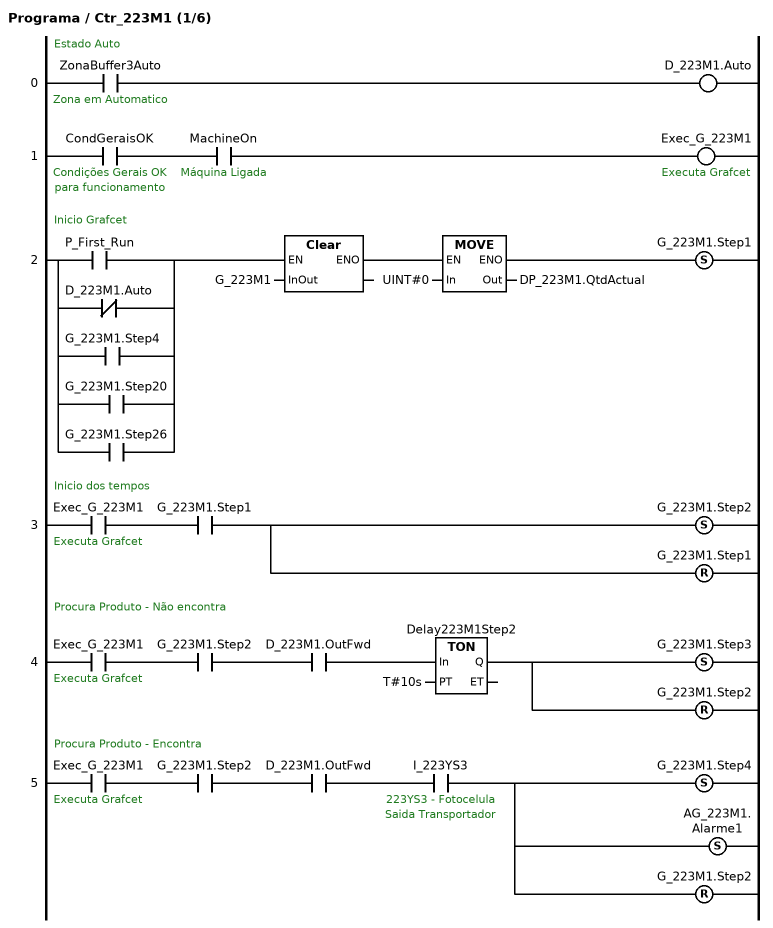
(* Rung 0: Estado Auto *)
D_223M1.Auto := ZonaBuffer3Auto;
(* Rung 1 *)
Exec_G_223M1 := CondGeraisOK AND MachineOn;
(* Rung 2: Inicio Grafcet *)
_p117 := P_First_Run OR NOT D_223M1.Auto OR G_223M1.Step4 OR G_223M1.Step20 OR G_223M1.Step26;
IF _p117 THEN
    Clear(InOut := G_223M1);
    DP_223M1.QtdActual := UINT#0;
    G_223M1.Step1 := TRUE;
END_IF;
(* Rung 3: Inicio dos tempos *)
_p118 := Exec_G_223M1 AND G_223M1.Step1;
IF _p118 THEN
    G_223M1.Step2 := TRUE;
    G_223M1.Step1 := FALSE;
END_IF;
(* Rung 4: Procura Produto - Não encontra *)
Delay223M1Step2(In := Exec_G_223M1 AND G_223M1.Step2 AND D_223M1.OutFwd, PT := T#10s);
IF Delay223M1Step2.Q THEN
    G_223M1.Step3 := TRUE;
    G_223M1.Step2 := FALSE;
END_IF;
(* Rung 5: Procura Produto - Encontra *)
_p119 := Exec_G_223M1 AND G_223M1.Step2 AND D_223M1.OutFwd AND I_223YS3;
IF _p119 THEN
    G_223M1.Step4 := TRUE;
    AG_223M1.Alarme1 := TRUE;
    G_223M1.Step2 := FALSE;
END_IF;

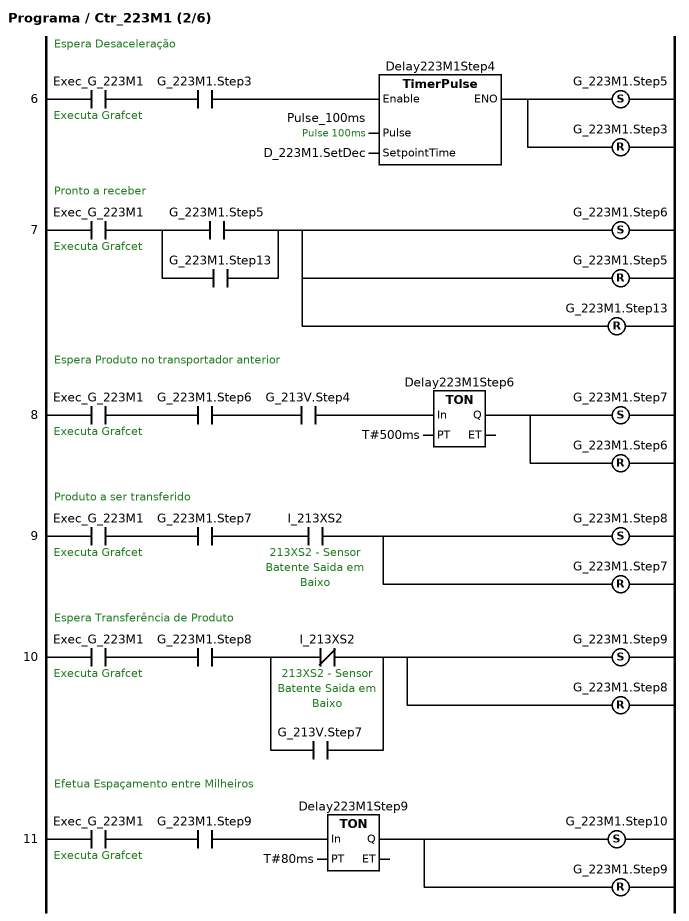
(* Rung 6: Espera Desaceleração *)
Delay223M1Step4(Enable := Exec_G_223M1 AND G_223M1.Step3, Pulse := Pulse_100ms, SetpointTime := D_223M1.SetDec);
IF Delay223M1Step4.ENO THEN
    G_223M1.Step5 := TRUE;
    G_223M1.Step3 := FALSE;
END_IF;
(* Rung 7: Pronto a receber *)
_p120 := Exec_G_223M1 AND (G_223M1.Step5 OR G_223M1.Step13);
IF _p120 THEN
    G_223M1.Step6 := TRUE;
    G_223M1.Step5 := FALSE;
    G_223M1.Step13 := FALSE;
END_IF;
(* Rung 8: Espera Produto no transportador anterior *)
Delay223M1Step6(In := Exec_G_223M1 AND G_223M1.Step6 AND G_213V.Step4, PT := T#500ms);
IF Delay223M1Step6.Q THEN
    G_223M1.Step7 := TRUE;
    G_223M1.Step6 := FALSE;
END_IF;
(* Rung 9: Produto a ser transferido *)
_p121 := Exec_G_223M1 AND G_223M1.Step7 AND I_213XS2;
IF _p121 THEN
    G_223M1.Step8 := TRUE;
    G_223M1.Step7 := FALSE;
END_IF;
(* Rung 10: Espera Transferência de Produto *)
_p122 := Exec_G_223M1 AND G_223M1.Step8 AND (NOT I_213XS2 OR G_213V.Step7);
IF _p122 THEN
    G_223M1.Step9 := TRUE;
    G_223M1.Step8 := FALSE;
END_IF;
(* Rung 11: Efetua Espaçamento entre Milheiros *)
Delay223M1Step9(In := Exec_G_223M1 AND G_223M1.Step9, PT := T#80ms);
IF Delay223M1Step9.Q THEN
    G_223M1.Step10 := TRUE;
    G_223M1.Step9 := FALSE;
END_IF;

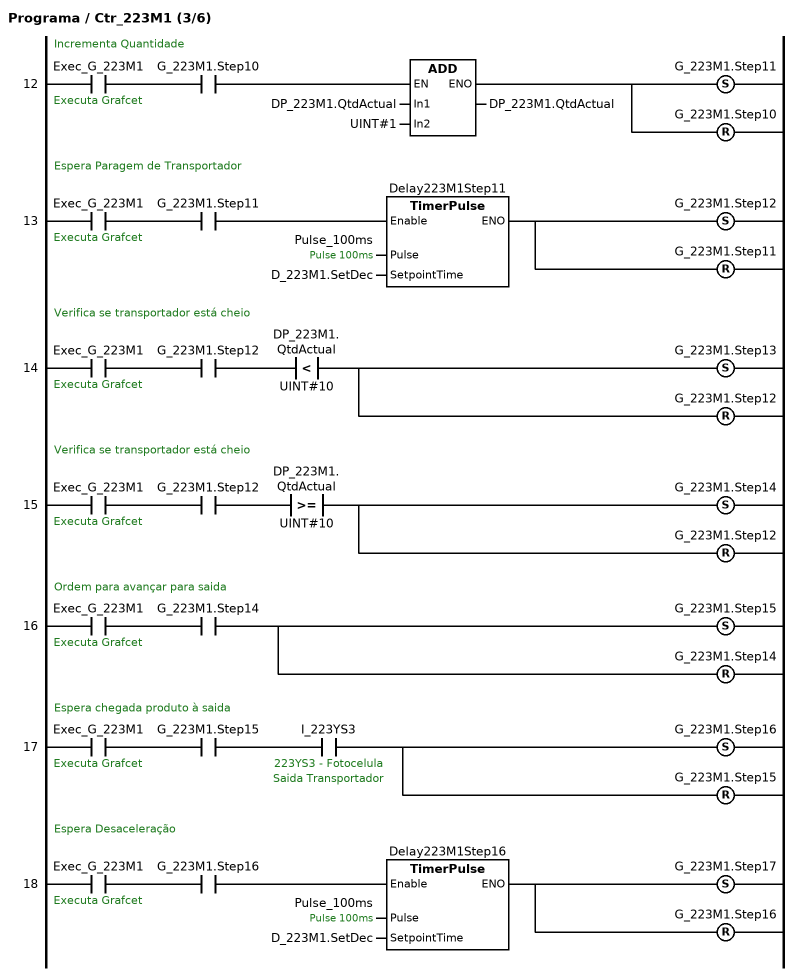
(* Rung 12: Incrementa Quantidade *)
IF Exec_G_223M1 AND G_223M1.Step10 THEN DP_223M1.QtdActual := DP_223M1.QtdActual + UINT#1; END_IF;
_p123 := Exec_G_223M1 AND G_223M1.Step10;
IF _p123 THEN
    G_223M1.Step11 := TRUE;
    G_223M1.Step10 := FALSE;
END_IF;
(* Rung 13: Espera Paragem de Transportador *)
Delay223M1Step11(Enable := Exec_G_223M1 AND G_223M1.Step11, Pulse := Pulse_100ms, SetpointTime := D_223M1.SetDec);
IF Delay223M1Step11.ENO THEN
    G_223M1.Step12 := TRUE;
    G_223M1.Step11 := FALSE;
END_IF;
(* Rung 14: Verifica se transportador está cheio *)
_p124 := Exec_G_223M1 AND G_223M1.Step12 AND (DP_223M1.QtdActual < UINT#10);
IF _p124 THEN
    G_223M1.Step13 := TRUE;
    G_223M1.Step12 := FALSE;
END_IF;
(* Rung 15: Verifica se transportador está cheio *)
_p125 := Exec_G_223M1 AND G_223M1.Step12 AND (DP_223M1.QtdActual >= UINT#10);
IF _p125 THEN
    G_223M1.Step14 := TRUE;
    G_223M1.Step12 := FALSE;
END_IF;
(* Rung 16: Ordem para avançar para saida *)
_p126 := Exec_G_223M1 AND G_223M1.Step14;
IF _p126 THEN
    G_223M1.Step15 := TRUE;
    G_223M1.Step14 := FALSE;
END_IF;
(* Rung 17: Espera chegada produto à saida *)
_p127 := Exec_G_223M1 AND G_223M1.Step15 AND I_223YS3;
IF _p127 THEN
    G_223M1.Step16 := TRUE;
    G_223M1.Step15 := FALSE;
END_IF;
(* Rung 18: Espera Desaceleração *)
Delay223M1Step16(Enable := Exec_G_223M1 AND G_223M1.Step16, Pulse := Pulse_100ms, SetpointTime := D_223M1.SetDec);
IF Delay223M1Step16.ENO THEN
    G_223M1.Step17 := TRUE;
    G_223M1.Step16 := FALSE;
END_IF;

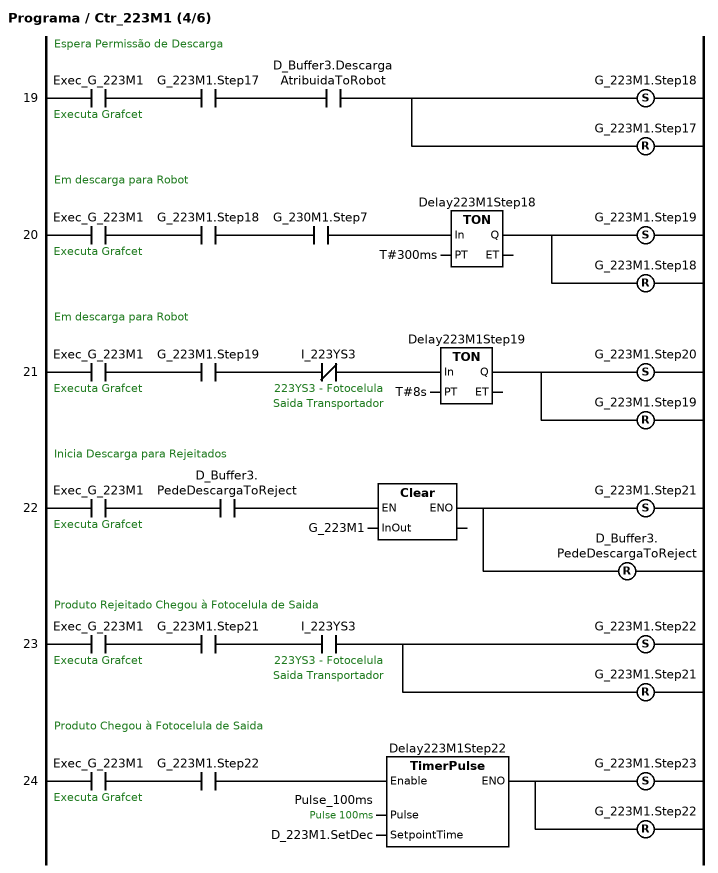
(* Rung 19: Espera Permissão de Descarga *)
_p128 := Exec_G_223M1 AND G_223M1.Step17 AND D_Buffer3.DescargaAtribuidaToRobot;
IF _p128 THEN
    G_223M1.Step18 := TRUE;
    G_223M1.Step17 := FALSE;
END_IF;
(* Rung 20: Em descarga para Robot *)
Delay223M1Step18(In := Exec_G_223M1 AND G_223M1.Step18 AND G_230M1.Step7, PT := T#300ms);
IF Delay223M1Step18.Q THEN
    G_223M1.Step19 := TRUE;
    G_223M1.Step18 := FALSE;
END_IF;
(* Rung 21: Em descarga para Robot *)
Delay223M1Step19(In := Exec_G_223M1 AND G_223M1.Step19 AND NOT I_223YS3, PT := T#8s);
IF Delay223M1Step19.Q THEN
    G_223M1.Step20 := TRUE;
    G_223M1.Step19 := FALSE;
END_IF;
(* Rung 22: Inicia Descarga para Rejeitados *)
IF Exec_G_223M1 AND D_Buffer3.PedeDescargaToReject THEN
    Clear(InOut := G_223M1);
    G_223M1.Step21 := TRUE;
    D_Buffer3.PedeDescargaToReject := FALSE;
END_IF;
(* Rung 23: Produto Rejeitado Chegou à Fotocelula de Saida *)
_p129 := Exec_G_223M1 AND G_223M1.Step21 AND I_223YS3;
IF _p129 THEN
    G_223M1.Step22 := TRUE;
    G_223M1.Step21 := FALSE;
END_IF;
(* Rung 24: Produto Chegou à Fotocelula de Saida *)
Delay223M1Step22(Enable := Exec_G_223M1 AND G_223M1.Step22, Pulse := Pulse_100ms, SetpointTime := D_223M1.SetDec);
IF Delay223M1Step22.ENO THEN
    G_223M1.Step23 := TRUE;
    G_223M1.Step22 := FALSE;
END_IF;

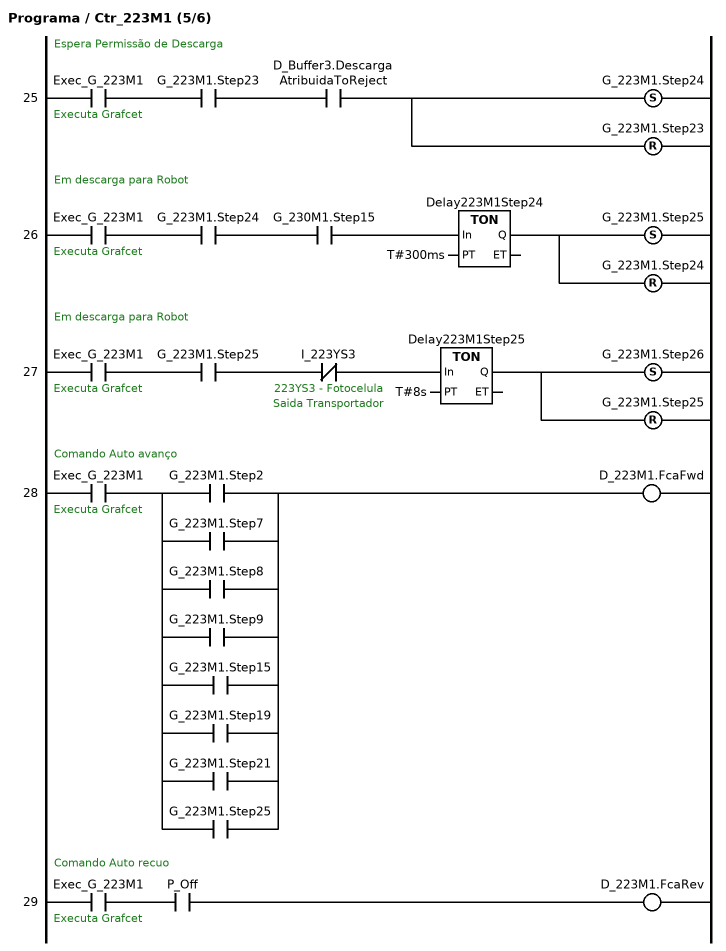
(* Rung 25: Espera Permissão de Descarga *)
_p130 := Exec_G_223M1 AND G_223M1.Step23 AND D_Buffer3.DescargaAtribuidaToReject;
IF _p130 THEN
    G_223M1.Step24 := TRUE;
    G_223M1.Step23 := FALSE;
END_IF;
(* Rung 26: Em descarga para Robot *)
Delay223M1Step24(In := Exec_G_223M1 AND G_223M1.Step24 AND G_230M1.Step15, PT := T#300ms);
IF Delay223M1Step24.Q THEN
    G_223M1.Step25 := TRUE;
    G_223M1.Step24 := FALSE;
END_IF;
(* Rung 27: Em descarga para Robot *)
Delay223M1Step25(In := Exec_G_223M1 AND G_223M1.Step25 AND NOT I_223YS3, PT := T#8s);
IF Delay223M1Step25.Q THEN
    G_223M1.Step26 := TRUE;
    G_223M1.Step25 := FALSE;
END_IF;
(* Rung 28: Comando Auto avanço *)
D_223M1.FcaFwd := Exec_G_223M1 AND (G_223M1.Step2 OR G_223M1.Step7 OR G_223M1.Step8 OR G_223M1.Step9 OR G_223M1.Step15 OR G_223M1.Step19 OR G_223M1.Step21 OR G_223M1.Step25);
(* Rung 29: Comando Auto recuo *)
D_223M1.FcaRev := Exec_G_223M1 AND P_Off;

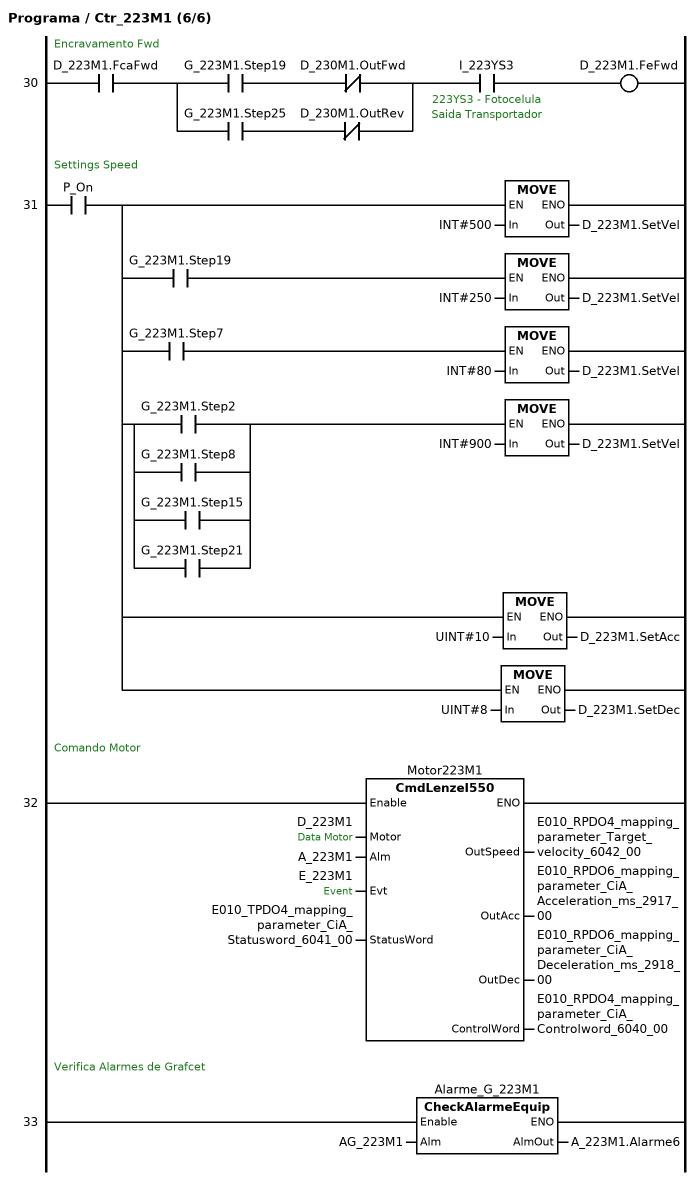
(* Rung 30: Encravamento Fwd *)
D_223M1.FeFwd := D_223M1.FcaFwd AND ((G_223M1.Step19 AND NOT D_230M1.OutFwd) OR (G_223M1.Step25 AND NOT D_230M1.OutRev)) AND I_223YS3;
(* Rung 31: Settings Speed *)
IF P_On THEN D_223M1.SetVel := INT#500; END_IF;
IF P_On AND G_223M1.Step19 THEN D_223M1.SetVel := INT#250; END_IF;
IF P_On AND G_223M1.Step7 THEN D_223M1.SetVel := INT#80; END_IF;
IF P_On AND (G_223M1.Step2 OR G_223M1.Step8 OR G_223M1.Step15 OR G_223M1.Step21) THEN
    D_223M1.SetVel := INT#900;
END_IF;
IF P_On THEN
    D_223M1.SetAcc := UINT#10;
    D_223M1.SetDec := UINT#8;
END_IF;
(* Rung 32: Comando Motor *)
Motor223M1(Enable := TRUE, Motor := D_223M1, Alm := A_223M1, Evt := E_223M1, StatusWord := E010_TPDO4_mapping_parameter_CiA_Statusword_6041_00, OutSpeed => E010_RPDO4_mapping_parameter_Target_velocity_6042_00, OutAcc => E010_RPDO6_mapping_parameter_CiA_Acceleration_ms_2917_00, OutDec => E010_RPDO6_mapping_parameter_CiA_Deceleration_ms_2918_00, ControlWord => E010_RPDO4_mapping_parameter_CiA_Controlword_6040_00);
(* Rung 33: Verifica Alarmes de Grafcet *)
Alarme_G_223M1(Enable := TRUE, Alm := AG_223M1, AlmOut => A_223M1.Alarme6);

(* Section Ctr_230M1: ladder, written here as Structured Text *)

